(*
Nazwa:			FB_CapPusherFeeder
Opis:			Sorter wibracyjny z rękawem
Wersja:			v1.0
Data:			2025-11-17
Autor:			DP
Urzadzenia:		Wkbracje, Wydmuch, czujniki zapełnienia rękawa
Konfiguracja:	
Info:
-
*)


FUNCTION_BLOCK FB_CapPusherFeeder
VAR_INPUT	
	bEnable						: BOOL;					//Zezowlenie na pracę stacji sprawdzania
	bEStop						: BOOL;					//Stop Awaryjny nieaktywny
	bRun						: BOOL;					//
	bHoming						: BOOL;					//Zezwolenie na wykonanie bazowania i pozycjonowania stacji sprawdzania
	bHeightSet					: BOOL;					//Bit do bazowania stacji na ustaloną wysokość 
	bIgnoreError				: BOOL;					//Ignorowania błędów cyklu pracy
	bReset						: BOOL;					//Reset błędu, jeśli w stanie "eError"

	bConveyorOKSensor			: BOOL;					
	bConveyorNOKSensor			: BOOL;				
	bAirOKSensor				: BOOL;					// 

	bCapsHopperSensor			: BOOL;					// Czujnik poziomu
	bCapsWheelSensor			: BOOL;					// Czujnik poziomu
	bCapsSleeveSensor			: BOOL;					// 
	bCapsSensor					: BOOL;

	iTimeDelayOn				: INT; 					//Czas na właczenie silnika sortera po zaniku sygnału przepełnienia z rękawa
	iTimeDelayOff				: INT; 					// Czas na wylączenie silnika sortera po wykryciu sygnału przepełnienia z rękawa sortera
	iTimeToEmptySleeveError		: INT;					// Czas do włączenia alrmu pustego rękawa
	InEngineVelocityCV 			: UDINT;		
	InEngineSTW 				: UINT; 				// Statusword transportera wejściowo wyjściowego
	IbEngineWcState				: BOOL; 				// Statusword transportera wejściowo wyjściowego

	bManualMovement				: BOOL; 				//Uruchomienie trybu ruchów ręcznych
	udiStationIndex				: UDINT;				// Indywidualny numer stacji
	sStationName				: WSTRING;				// Nazwa stacji	
END_VAR

VAR_OUTPUT
	eState						: E_Station;			// Aktualny stan stacju
	eRunningState				: E_CapFeederState;		// Stan pracy stacji
	bError						: BOOL;					// Błąd stacji
	udiErrorID					: UDINT;				// Nr blędu przeciągania formatek
	sErrorDescription			: STRING(200);			// Opis błędu
	sErrorDescription2			: STRING(200);			// Opis błędu
	sErrorStationName			: STRING;				// Nazwa stacj
	udiStationID				: UDINT;				// Nr stacji

	QnEngineVelocitySV 			: UDINT; 				// Nastawa prędkości
	QnEngineCTW 				: UINT;  				// Controlword transportera we/wy	
	bSorterVibrator				: BOOL; 	
	bSorterVibrator2			: BOOL; 	
	bSorterAir 					: BOOL; 							
	
	bHomingNeeded				: BOOL;					// Wymagane ponowne bazowanie (blad podczas bazowania lub stop awaryjny)
	bHomingDone					: BOOL;					// Stacja zbazowana 
	bCycleDone					: BOOL;					// Sygnał o zakończeniu cyklu
	bCycleNotDone				: BOOL;					// Sygnał o niezakończonym cyklu
	tCycleTime					: TIME;	 				// Czas cyklu 
	sWarningDescription			: STRING;
	bWarning1					: BOOL;
	udiWarningID				: UDINT;
END_VAR

VAR_IN_OUT
	bManualSorterEngine			: BOOL;					//
	bManualSorterVibrator		: BOOL;					//
	bManualSorterVibrator2		: BOOL;					//
	bManualSorterAir 			: BOOL;					//
END_VAR

VAR
	i							:	INT;

	// State
	eLastState					: E_Station;			//Stan ogólny bloku
	eLastStateTemp				: E_Station;			//Stan ogólny bloku
	eLastRunningState			: E_CapFeederState;		//Stan podbloku
	eLastRunningStateTemp		: E_CapFeederState;		//Stan podbloku

	bStateError					: BOOL;
		
	tonSortingEngineOn			: TON;					// Opóźnienie po załączeniu napędu
	tonSortingEngineOff			: TON;					// Opóźnienie wyłączenia napędu
	tonAirBeforeStart			: TON;					// Czasówka opóźeniani przedmuchu
	tonAirAfterStop				: TON;					// Czasówka przedmuchu po zatrzymaniu
	tonStoppingTime				: TON;					// Czasówka zbyt długiego zatrzymawania

	tonEmptySleeveError			: TON;					// Timer pustego rękawa
	tonCycleTimer				: TON;					// Czasówka cyklu
	rtrigCycleTimerRead			: R_TRIG;				// Trigger do statystyk cyklu 
	
	fbInverter: FB_MitsubishiInverter;
	tonInverterError: TON;
	tonAirError: TON;
	(*Ostrzeżenia*)
	fbbLevelSensor:	FB_InputFilter_v2;
	(*Inne*)	
	fbbCapsWheelLevelSensor 		: FB_InputFilter_v2;
	fbbCapsAndSleeveSensor			: FB_InputFilter_v2;
	tonVibrator2AndNotbCapsSensor	: TON;
	tonbSorterVibrator				: TON;
	tonfbInverterbRun1				: TON;
	tonfbInverterbRun2				: TON;	
	//Zmienne od EVENTLOGGER
	bAlarmInit 						: BOOL := TRUE; 
	nAlarmNumerator					: INT;
	arfbAlarm						: ARRAY[0..19] OF  FB_TcAlarm;		//Tablica bloczków błędów
	fbSourceInfo 					: FB_TcSourceInfo;
	iSourceInfo						: I_TcSourceInfo;
	sAlarmTest						: STRING;
	//Koniec zmiennych od EVENTLOGGER
	iSortingCASE					: INT;
	tonNoCapsHopperSensor			: TON;
END_VAR

//Wywołanie bloczków od stacji. Ważna jest ich kolejność!!!
ACT_Limits();
ACT_ErrorHandling();
ACT_Signals();
ACT_Control();
ACT_Inverter();
ACT_Statistic();
ACT_Status();
ACT_Warnings();
aStationID();

ACTION ACT_Control:
	(*****Wyłączenie enable*****)
	IF NOT bEnable THEN
		IF eState <> E_Station.eDisabled AND eState <> E_Station.ePreparingToDisable THEN
				eState 				:= E_Station.ePreparingToDisable; 
		END_IF	
	END_IF

	(*****Estop*****)
	IF NOT bEstop  THEN	
		IF eState <> E_Station.eAborted AND eState <> E_Station.eAborting AND eState <> E_Station.eDisabled THEN
				eState 				:= E_Station.eAborting; 
		END_IF
	END_IF

	CASE eState OF
//--------------------------------------------------------------------------------
// Stan maszyny po wyłączeniu i przygotowanie do uruchomienia
	E_Station.eDisabled: 					// Stan nieaktywnosci (Stacja wyłączona) 
	
		IF bEnable THEN
			eState 				:= E_Station.ePreparingToReady; 
		END_IF 
		
//--------------------------------------------------------------------------------
// Stan maszyny po zatrzymaniu awaryjnym   
	E_Station.eAborted: 					// Stan bezpiecznego zatrzymania (po Abortingu) 

		IF bEStop THEN
			eState 				:= E_Station.ePreparingToReady;
		END_IF
		
//--------------------------------------------------------------------------------
// Stan maszyny naciśnieciu estopa 	
	E_Station.eAborting:                 	// Stan bezpiecznego zatrzymywania (po EStopie)

		ACT_ResetCommands();

		eState 						:=  E_Station.eAborted;  
		eRunningState				:=	E_CapFeederState.eReady;
		
//--------------------------------------------------------------------------------
// Stan masyzny po wykryciu błędu			
	E_Station.eError:                 	 	// Stan błędu 	
		
		ACT_ResetCommands();
		
		IF bReset THEN
			eState 				:= E_Station.eResetting;
			bError				:= FALSE;
		END_IF
		
//--------------------------------------------------------------------------------
// Stan masyzny po wykryciu błędu
	E_Station.eResetting:					// Stan resetowania bledu (po Errorze)
		
			fbInverter.bReset	:= TRUE;
		IF NOT bError (*AND fbInverter.eState = E_Station.eReady*) THEN
			fbInverter.bReset	:= FALSE;	
			//{warning 'Sprawdzić błąd falownika CapFeeder'}
			udiErrorID 			:=	0;
			sErrorDescription 	:=	'';
			eState 				:=	E_Station.ePreparingToReady;
			eRunningState		:=	E_CapFeederState.eReady;
		ELSE
			eState 				:=	E_Station.eError;
		END_IF
    
//--------------------------------------------------------------------------------
// Stan ruchoow manualnych
	E_Station.eManualMovement:     			// Stan ruchów manualnych  
   
		ACT_ManualMovements();
		//Wyjście z trybu serwisowego
		IF NOT bManualMovement THEN		
			eState:=E_Station.eReady;
		END_IF
		

//--------------------------------------------------------------------------------
// Stan rozpoczecia bazowania
	E_Station.eHoming:						// Stan bazowania 
		
		ACT_Homing();
		IF NOT bHoming AND NOT bHeightSet THEN
		   eState								:=	E_Station.ePreparingToReady;
		END_IF		
		
//--------------------------------------------------------------------------------
// Stan zakończenia bazowania
	E_Station.eHomingDone:                  // Stan wykonania bazowania 
	
		bHomingDone							:=	TRUE;
		IF NOT bHoming AND NOT bHeightSet THEN
		   eState:=E_Station.eReady;
		END_IF
		
//--------------------------------------------------------------------------------
// Stan przygotowania do gotowości
	E_Station.ePreparingToReady:            // Stan przygotowywania do gotowosci (zawsze przed Ready)  
		
		fbInverter.bRun						:=	FALSE;
		bSorterAir							:=	FALSE;
		bSorterVibrator						:=	FALSE;
		bSorterVibrator2					:=	FALSE;

		eRunningState						:=	E_CapFeederState.eReady;
		eState								:=	E_Station.eReady;	
		
//-------------------------------------------------------------------------------
// Stan przygotowania do wyłączenia maszyny
	E_Station.ePreparingToDisable:          // Stan przygotowywania do nieaktywnosci (po wyłączeniu Enable) 
		
		bSorterAir							:=	FALSE;

		eRunningState						:=	E_CapFeederState.eReady;		
		eState								:=	E_Station.eDisabled;

			
//--------------------------------------------------------------------------------
// Stan gotowości
	E_Station.eReady:						// Stan gotowosci 

		IF bRun AND NOT bCycleDone AND NOT bCycleNotDone THEN
			eState 							:= E_Station.eStarting; 
		END_IF
		IF bHoming OR bHeightSet THEN
			bHomingDone						:=	FALSE;
			eState 							:=	E_Station.eHoming; 
		END_IF
		IF bManualMovement THEN
			//Jeśli przejście w tryb ruchów manualnych przepisz wszystkie stany siłowników sterowanych przez moduł
			//aby zapobiec ewentualnym kolizjom po wejściu w tryb serwisowy
			eState 						:= E_Station.eManualMovement; 
		END_IF
		IF NOT bRun THEN
			bCycleDone 			:= FALSE;
			bCycleNotDone 		:= FALSE;			
		END_IF
		
//--------------------------------------------------------------------------------
// Stan zatrzymywania
	E_Station.eStopping:					// Stan zatrzymywania 
		
	bSorterVibrator	:=	FALSE;
	bSorterVibrator2:=	FALSE;
	bSorterAir		:=	TRUE;
	fbInverter.bRun := FALSE;
	
	IF tonStoppingTime.Q THEN
		ACT_ResetCommands();
		eRunningState							:= E_CapFeederState.eReady;
		eState									:= E_Station.eReady;
	END_IF
		
//--------------------------------------------------------------------------------
// Stan uruchomienia lini ( po eReady)
	E_Station.eStarting:                  	// Stan uruchamiania (po Ready)

		eState					 := E_Station.eRunning; 
		
//--------------------------------------------------------------------------------
// Stan wykonywania pracy
	E_Station.eRunning:               		// Stan wykonywania cyklu (po Startingu), w tym stanie osobny

		ACT_Running();
		IF NOT bRun THEN 					(*Przerywanie cyklu*)
			eState				:= E_Station.eStopping;
			//bCycleNotDone		:= TRUE;
		END_IF
		(*IF bCycleDone OR bCycleNotDone THEN (*Cykl zakończony*)
			eState 				 := E_Station.eReady;
		END_IF*)							
		
END_CASE
END_ACTION

ACTION ACT_ErrorHandling:
// Alarm_0600	600	Error	Pusty rekaw wbijaka nasadek - sprawdź czy nasadki sie nie zablokowały
// Alarm_0601	601	Error	Błąd falownika - możliwe zablokowanie mechaniczne transportera
// Alarm_0602	602	Error	Bład czujnika powietrza - sprwadź ciśnienie

IF bAlarmInit THEN
    bAlarmInit := FALSE; 
	fbSourceInfo.Clear();
	fbSourceInfo.sName:=wsLiteral_TO_UTF8(sStationName);//'Machine';
	fbSourceInfo.nId:=udiStationID;//2700;
	// Alarm_0600	600	Error	Pusty rekaw wbijaka nasadek - sprawdź czy nasadki sie nie zablokowały
    arfbAlarm[0].CreateEx(stEventEntry := TC_EVENTS.AlarmClass.Alarm_0600, bWithConfirmation:= FALSE,  ipSourceInfo:= fbSourceInfo); 
	// Alarm_0601	601	Error	Błąd falownika - możliwe zablokowanie mechaniczne transportera
	arfbAlarm[1].CreateEx(stEventEntry := TC_EVENTS.AlarmClass.Alarm_0601, bWithConfirmation:= FALSE,  ipSourceInfo:= fbSourceInfo);
	// Alarm_0602	602	Error	Bład czujnika powietrza - sprwadź ciśnienie	
	arfbAlarm[2].CreateEx(stEventEntry := TC_EVENTS.AlarmClass.Alarm_0602, bWithConfirmation:= FALSE,  ipSourceInfo:= fbSourceInfo);	
	// Alarm_0603	603	Error	Blokada nasadek przed wbijaniem - sprawdź czujnik
    arfbAlarm[3].CreateEx(stEventEntry := TC_EVENTS.AlarmClass.Alarm_0603, bWithConfirmation:= FALSE,  ipSourceInfo:= fbSourceInfo);  
	// Alarm_0604	604	Error	Brak nakrętek w zbiorniku
    arfbAlarm[4].CreateEx(stEventEntry := TC_EVENTS.AlarmClass.Alarm_0604, bWithConfirmation:= FALSE,  ipSourceInfo:= fbSourceInfo);	{warning 'Zmienić opis alarmu powyżej po dodaniu do listy'}
END_IF

//OBSŁUGA BŁĘDÓW STACJI SPRAWDZANIA
//************LISTA BŁĘDÓW***************
bStateError:= (eState=E_Station.eError) OR (eState=E_Station.eResetting);

//************LISTA BŁĘDÓW***************

//Error 1 - podnośnik nie porusza się pomimo wysterowania 
tonEmptySleeveError				(IN:=NOT bCapsSleeveSensor AND bRun, PT:=INT_TO_TIME(iTimeToEmptySleeveError)*1000); //Było 30, teraz jest z receptur
tonInverterError				(IN:=fbInverter.bError AND NOT bStateError, PT:=T#3S);
tonAirError						(IN:=bSorterAir AND NOT bAirOKSensor AND NOT bStateError, PT:=T#3S);
tonVibrator2AndNotbCapsSensor	(IN:=bSorterVibrator2 AND fbbCapsWheelLevelSensor.bOut AND  NOT bCapsSensor AND P07_CapPusher.fbCapPusherFeeder.eState = E_Station.eRunning, PT:=T#30S);
tonNoCapsHopperSensor			(IN:= NOT bCapsHopperSensor AND P07_CapPusher.fbCapPusherFeeder.eState = E_Station.eRunning AND NOT VIS.bConfectionEnding, PT:=T#30S);

IF (bEnable OR (eState = E_Station.ePreparingToDisable)) THEN
	
		
	//Error - Pusty rekaw sortera nasadek
	IF tonEmptySleeveError.Q THEN
		IF NOT arfbAlarm[0].bActive THEN
			arfbAlarm[0].Raise(nTimeStamp:=0);
		END_IF
	ELSE	
		IF  arfbAlarm[0].bActive AND bReset THEN
			arfbAlarm[0].Clear(nTimeStamp:=0, bResetConfirmation:= FALSE);
		END_IF
	END_IF	
		
	//Error - Bład falownika
	IF tonInverterError.Q THEN
		IF NOT arfbAlarm[1].bActive THEN
			arfbAlarm[1].Raise(nTimeStamp:=0);
		END_IF
	ELSE	
		IF  arfbAlarm[1].bActive AND bReset THEN
			arfbAlarm[1].Clear(nTimeStamp:=0, bResetConfirmation:= FALSE);
		END_IF
	END_IF		
	
	//Error - Bład powietrza
	IF tonAirError.Q THEN
		IF NOT arfbAlarm[2].bActive THEN
			arfbAlarm[2].Raise(nTimeStamp:=0);
		END_IF
	ELSE	
		IF  arfbAlarm[2].bActive AND bReset THEN
			arfbAlarm[2].Clear(nTimeStamp:=0, bResetConfirmation:= FALSE);
		END_IF
	END_IF		
	
	//Error - Nakrętki nie dojechały do czujnika nad butelka
	IF tonVibrator2AndNotbCapsSensor.Q THEN
		IF NOT arfbAlarm[3].bActive THEN
			arfbAlarm[3].Raise(nTimeStamp:=0);
		END_IF
	ELSE	
		IF  arfbAlarm[3].bActive AND bReset THEN
			arfbAlarm[3].Clear(nTimeStamp:=0, bResetConfirmation:= FALSE);
		END_IF
	END_IF		
	
	//Error - Brak nakrętek w zbiorniku
	IF tonNoCapsHopperSensor.Q THEN
		IF NOT arfbAlarm[4].bActive THEN
			arfbAlarm[4].Raise(nTimeStamp:=0);
		END_IF
	ELSE	
		IF  arfbAlarm[4].bActive AND bReset THEN
			arfbAlarm[4].Clear(nTimeStamp:=0, bResetConfirmation:= FALSE);
		END_IF
	END_IF			
ELSE
	bError	:=FALSE;
		IF  arfbAlarm[0].bActive THEN
			arfbAlarm[0].Clear(nTimeStamp:=0, bResetConfirmation:= FALSE);
		END_IF
		IF  arfbAlarm[1].bActive THEN
			arfbAlarm[1].Clear(nTimeStamp:=0, bResetConfirmation:= FALSE);
		END_IF
		IF  arfbAlarm[2].bActive THEN
			arfbAlarm[2].Clear(nTimeStamp:=0, bResetConfirmation:= FALSE);
		END_IF
		IF  arfbAlarm[3].bActive THEN
			arfbAlarm[3].Clear(nTimeStamp:=0, bResetConfirmation:= FALSE);
		END_IF
		IF  arfbAlarm[4].bActive THEN
			arfbAlarm[4].Clear(nTimeStamp:=0, bResetConfirmation:= FALSE);
		END_IF	
END_IF


//-----------------------------------------------------------------------
IF bError AND NOT bStateError THEN

	IF eLastState = eRunning THEN
		bCycleNotDone						:= TRUE;
	END_IF
	eState 									:= E_Station.eError;
END_IF

//------------------------------------------------------------------------
(*Wyświetlanie błedu na wyjściu*)
bError							:= FALSE;
FOR nAlarmNumerator := 0 TO 19 DO
	bError						:= bError OR arfbAlarm[nAlarmNumerator].bActive;
END_FOR

(*Wyświetlanie błedu na wyjściu*)
bError;

(*Przepisywanie nazwy stacji*)
sErrorStationName 							:= WSTRING_TO_STRING(sStationName);
END_ACTION

ACTION ACT_Homing:
//BAZOWANIE
eState:=E_Station.eHomingDone;
END_ACTION

ACTION ACT_Inverter:
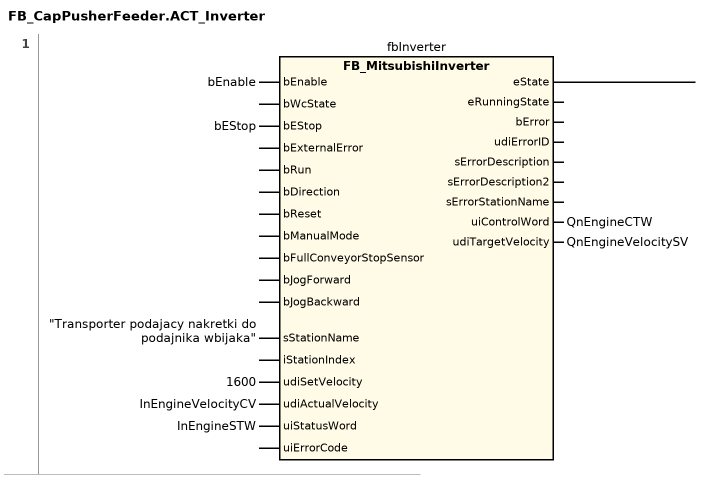
// NETWORK 1
fbInverter(
    bEnable := bEnable,
    bEStop := bEStop,
    sStationName := "Transporter podajacy nakretki do podajnika wbijaka",
    udiSetVelocity := 1600,
    udiActualVelocity := InEngineVelocityCV,
    uiStatusWord := InEngineSTW,
    uiControlWord => QnEngineCTW,
    udiTargetVelocity => QnEngineVelocitySV); // FB_MitsubishiInverter
END_ACTION

ACTION ACT_Limits:
IF iTimeToEmptySleeveError < 5 THEN
	iTimeToEmptySleeveError := 5;
END_IF
END_ACTION

ACTION ACT_ManualMovements:
//W trybie ruchów manualnych wykonuj ruchy za pomocą rozkazów manualnych
IF NOT bRun THEN
	fbInverter.bRun		:= bManualSorterEngine;
	bSorterVibrator		:= bManualSorterVibrator;
	bSorterVibrator2	:= bManualSorterVibrator2;	
	bSorterAir			:= bManualSorterAir;
END_IF

IF bHoming OR bHeightSet THEN
	eState:=E_Station.eHoming;
END_IF

IF bRun THEN	
	ACT_Running();
END_IF
//Zabezpieczenie przed kolizją stacji poprzez ruch podnośnika
END_ACTION

ACTION ACT_ResetCommands:
//Reset komend ruchu 	

fbInverter.bRun	:=	FALSE;
bSorterAir		:=	FALSE;
bSorterVibrator	:=	FALSE;
bSorterVibrator2:=	FALSE;
END_ACTION

ACTION ACT_Running:
//----------------------------------------------------------------------------------
// Obsługa podajnik zamknięc

CASE eRunningState OF
	
	//NIEGOTOWY
	E_CapFeederState.eDisabled:
		eRunningState			:=	E_CapFeederState.eReady;

	E_CapFeederState.eReady:
		fbInverter.bDirection 	:=	FALSE;
		IF bRun THEN
			iSortingCASE		:= 0;
			eRunningState		:=	E_CapFeederState.eSorting;
		END_IF
	
	E_CapFeederState.eSorting:
	
		// 	1-Najpierw powietrze
		//	2-Potem wibracje rekawa
		//	3-Potem wibracje kola jezeli nie ma na czujniku
		bSorterAir 				:= TRUE;			
		bSorterVibrator 		:= tonAirBeforeStart.Q;
		bSorterVibrator2 		:= TRUE;
		fbInverter.bRun 		:= fbbCapsWheelLevelSensor.bOut AND tonbSorterVibrator.Q ;
		
		CASE iSortingCASE OF 
			0:
				iSortingCASE			:=	iSortingCASE	+	10;
			
			10:
				fbInverter.bRun 		:= fbbCapsWheelLevelSensor.bOut AND tonbSorterVibrator.Q ;
				IF tonfbInverterbRun1.Q THEN //Chodzi 1s
					iSortingCASE		:=	iSortingCASE	+	10;
				END_IF
				
			20:
				fbInverter.bRun := FALSE;
				IF tonfbInverterbRun2.Q THEN //Stop 2s
					iSortingCASE	:=	10;
				END_IF
							
		END_CASE
			
		IF tonSortingEngineOff.Q THEN  //5S
			eRunningState 			:=E_CapFeederState.eSleeveFull;
		END_IF
	
	E_CapFeederState.eSleeveFull:
		bSorterVibrator 	:=	FALSE;		
		IF fbbCapsAndSleeveSensor.bOUT THEN
			bSorterVibrator2 	:= FALSE;
		ELSE
			bSorterVibrator2 	:= TRUE;
		END_IF
		fbInverter.bRun		:=	FALSE;
		bSorterAir			:=	NOT tonAirAfterStop.Q;
		IF tonAirAfterStop.Q THEN
			IF tonSortingEngineOn.Q THEN
				iSortingCASE		:= 0;
				eRunningState		:=E_CapFeederState.eSorting; 
			END_IF
		END_IF
	
	E_CapFeederState.eSleeveLowLevel:
	
		;
	
END_CASE
END_ACTION

ACTION ACT_Signals:
(** Timery na potrzeby bazowania**)
//Czujnik poziomu na kole
fbbCapsWheelLevelSensor		(bIN:=NOT bCapsWheelSensor AND eRunningState=E_CapFeederState.eSorting,		tFilterTimeOn:= T#8S, tFilterTimeOff:= T#40MS, bOUT=> );
fbbCapsWheelLevelSensor.bOut;

fbbCapsAndSleeveSensor		(bIN:=bCapsSleeveSensor AND bCapsSensor,		tFilterTimeOn:= T#2S, tFilterTimeOff:= T#100MS, bOUT=> );
tonbSorterVibrator			(IN:= bSorterVibrator, 					PT:=T#4S);
tonfbInverterbRun1			(IN:=fbInverter.bRun, 					PT:=T#600MS);
tonfbInverterbRun2			(IN:=NOT fbInverter.bRun, 				PT:=T#3S);


tonAirBeforeStart		(IN:=eRunningState=E_CapFeederState.eSorting, PT:=T#1S);
tonSortingEngineOff		(IN:=((eRunningState=E_CapFeederState.eSorting OR eRunningState=E_CapFeederState.eSleeveLowLevel) AND bRun AND bCapsSleeveSensor),PT:=INT_TO_TIME(iTimeDelayOff));
tonAirAfterStop			(IN:=eRunningState=E_CapFeederState.eSleeveFull, PT:=T#2S);
tonSortingEngineOn		(IN:=((eRunningState=E_CapFeederState.eSorting OR eRunningState=E_CapFeederState.eSleeveFull) AND bRun AND NOT bCapsSleeveSensor),PT:=INT_TO_TIME(iTimeDelayOn));
	
(** Timery używane podczas pracy stacji**)


(** Dodatkowy timer przy zatrzymywaniu**)
tonStoppingTime( IN:= eState= E_Station.eStopping, PT:=T#2S);
VIS_CP.IbCapPusher0DoorsOpen := NOT VIS_CP.IbCapPusher0DoorsOpen;
END_ACTION

ACTION ACT_Statistic:
//Statystyka do zliczania czasu cyklu 
rtrigCycleTimerRead(CLK:=eRunningState=E_CapFeederState.eSleeveFull OR eRunningState=E_CapFeederState.eSleeveLowLevel);

	IF rtrigCycleTimerRead.Q THEN
		tCycleTime:=tonCycleTimer.ET;
		
	END_IF
	
tonCycleTimer(IN:=eRunningState= E_CapFeederState.eSorting , PT:=T#1D);
END_ACTION

ACTION ACT_Status:

(*Zapisywanie ostatniego stanu*)
	IF eLastStateTemp<>eState THEN
		eLastState := eLastStateTemp;
	END_IF
	eLastStateTemp := eState;
	
	IF eLastRunningStateTemp<>eRunningState THEN
		eLastRunningState := eLastRunningStateTemp;
	END_IF
	eLastRunningStateTemp := eRunningState;
(*Koniec Zapisywanie ostatniego stanu*)
END_ACTION

ACTION ACT_Warnings:
//Usrawianie warningów

//Filtrowanie czujnika ultradźwiękowego
fbbLevelSensor	(bIN:=NOT bCapsSleeveSensor AND (eRunningState=E_CapFeederState.eSorting OR eRunningState=E_CapFeederState.eSleeveLowLevel OR eRunningState=E_CapFeederState.eSleeveFull) , tFilterTimeOn:= T#5S, tFilterTimeOff:=T#5S , bOUT=> );

IF fbbLevelSensor.bOUT THEN
		bWarning1						:=	TRUE;			
		udiWarningID					:=	1;
		sWarningDescription				:=	'Niski poziom w sorterze nasadek';
ELSE
		bWarning1						:=	FALSE;			
		udiWarningID					:=	0;
		sWarningDescription				:=	'';
END_IF
END_ACTION

ACTION aStationID:
udiStationID	:=	udiStationIndex;
END_ACTION

END_FUNCTION_BLOCK

(* stored: Version 1.2.0.0, ProductVersion 3.1.4026.13, FileIdentifier 59b20936cd15aaec5ba9f02cc006617b23940bf9, FileSignature 00e9870dcaa53f873610d463e4f2766c8110e98e08cecbeee3b57709a8eec143a7e389ec8915ae8199c7a49ae1a702fc2a4bd80a8f1130ed8730aa2fc9231f28527f6fb983ac45f505853f842ba00214cce7088f5ced859dc6c12ae50c3f92b4c86b5ffb968f375c76b15e5dc254754c5be139dc2d746e3dd5cbd6bbf45fb8cb524aab5d2fcfd1efb706dbc8541b4079cf56c5a20df83340bd105443b24cb7a1271d667084862781aedbbd25dc3d7bc620a629765c74bb48d86d0b432bbbe31305973631617960c7567907337eda4a1f8c1b54785636bba67562cd2254fb714edf58dcca7fc03af40545e3ca363be278a74a76ee6edfa6e67ba0dc799c7517a1
   POU FB_CapPusherFeeder: Id {1fed3b59-03fb-4d91-bd48-1fb0cd917150}, SpecialFunc None
   Action ACT_Control: Id {0587746b-7ce6-453a-9ea4-0327b7df915e}
   Action ACT_ErrorHandling: Id {6b0a3037-1437-4edd-b79e-1697981c6162}
   Action ACT_Homing: Id {43ec9bee-9915-445d-8d53-036099cc45a4}
   Action ACT_Inverter: Id {30f8a855-c4e3-499a-9107-cca6e690391d}
   Action ACT_Limits: Id {be8ed520-1fea-48d4-90a2-36250bfcbee8}
   Action ACT_ManualMovements: Id {28fee632-4c09-40ea-897c-d155c56b0fb2}
   Action ACT_ResetCommands: Id {74959fa6-c2c7-4d86-b586-a2964a0121cb}
   Action ACT_Running: Id {a25eb625-0563-4bff-b701-24633266cbd4}
   Action ACT_Signals: Id {0277d687-6a96-411b-9fd3-b105f95e7e85}
   Action ACT_Statistic: Id {b185a0f9-6be9-4710-85b8-97bcf5e6b0a7}
   Action ACT_Status: Id {28871896-75ed-4fc5-9730-1efe02717cbf}
   Action ACT_Warnings: Id {5062fbc9-4088-4718-8c9f-ef5849da15d9}
   Action aStationID: Id {7a82ca5a-c19b-41ef-886e-4b84264f381c} *)
